Universal Robots PolyScope program: track.urp

Program track (installation=default directory=/home/ur/ursim-current/programs createdIn=5.12.6.1102099 lastSavedIn=5.12.6.1102099 robotSerialNumber=20195299999)
Calibrated DH parameters: a=[0, -0.6127, -0.57155, 0, 0, 0]; d=[0.1807, 0, 0, 0.17415, 0.11985, 0.11655]; alpha=[1.570796, 0, 0, 1.570796, -1.570796, 0]; deltaTheta=[0, 0, 0, 0, 0, 0]
BeforeStart
  MoveJ speed 60 deg/s, acceleration 80 deg/s^2 (useActiveTCP=true) feature=Base
    Waypoint Waypoint_1: TCP in base x=-164.283 y=-550.453 z=498.391 mm, rx=0.0278 ry=-2.2221 rz=2.1846 rad; joints [-88.604, -92.965, -133.167, 45.162, 88.284, -1.724] deg
  x := 0.1
  z := 0.1
Robot Program (runOnlyOnce=false)
  If digital_out[0]≟ True (checkContinuously=true)
    Script: speedl([x,0,z,0,0,0],0.3,0.3)
  Else 
    Script: stopl(20.0)
Thread Thread_1 (runOnlyOnce=false)
  x := (320-x0)/1000
  z := (240-zo)/1000
